DATA_BLOCK "DB2006_SA"
TITLE = DB2006_SA
{ S7_Optimized_Access := 'FALSE' }
AUTHOR : ABH
FAMILY : ZeusControl
VERSION : 1.0
//Bloique de datos Salida Analogica
   STRUCT
      SA { S7_SetPoint := 'False'} : Array[0.."N_MAX_DISP_SA"] of "UDT_ZC_DISP_SA";
      Mux { S7_SetPoint := 'False'} : Array[0.."N_MAX_MUX_DISP"] of "UDT_ZC_DISP_MUX_SA";
      Agrup : Array[0.."N_MAX_DISP_AGRUP"] of "UDT_ZC_DISP_AGRUP";
   END_STRUCT;


BEGIN
   SA[0].Hmi_Estado := 0;
   SA[0].Estado_ValorIngenieria := 0.0;
   SA[0].Estado_AutoMan := FALSE;
   SA[0].Estado_Enclavado := FALSE;
   SA[0].Alarmas_Min := FALSE;
   SA[0].Alarmas_Max := FALSE;
   SA[0].Alarmas_Escritura := FALSE;
   SA[0].Alarmas_Parametros := FALSE;
   SA[0].Alarmas_General := FALSE;
   SA[0].Config_Habilitar := FALSE;
   SA[0].Config_HabilitarAlarmaMin := FALSE;
   SA[0].Config_HabilitarAlarmaMax := FALSE;
   SA[0].Aux_oldAlarma := FALSE;
   SA[0].Aux_oldAutoMan := FALSE;
   SA[0].Estado_SeguridadOk := TRUE;
   SA[0].Config_GrupoAlarma := 0;
   SA[0].Aux_Estado := 0;
   SA[0].Estado_ValorTarjeta := 0;
   SA[0].Estado_Escritura := 16#0000;
   SA[0].Orden_ConsignaManual := 0.0;
   SA[0].Orden_ConsignaAuto := 0.0;
   SA[0].Orden_ConsignaEnclavado := 0.0;
   SA[0].Config_DireccionSalidaByte := 0;
   SA[0].Config_EscaladoMinTarjeta := 0;
   SA[0].Config_EscaladoMaxTarjeta := 27648;
   SA[0].Config_EscaladoMinIngenieria := 0.0;
   SA[0].Config_EscaladoMaxIngenieria := 0.0;
   SA[0].Config_EscaladoOffset := 0.0;
   SA[0].Config_ErrorMinIngenieria := 0.0;
   SA[0].Config_ErrorMaxIngenieria := 0.0;
   SA[1].Hmi_Estado := 1;
   SA[1].Estado_ValorIngenieria := 0.0;
   SA[1].Estado_AutoMan := FALSE;
   SA[1].Estado_Enclavado := FALSE;
   SA[1].Alarmas_Min := FALSE;
   SA[1].Alarmas_Max := FALSE;
   SA[1].Alarmas_Escritura := FALSE;
   SA[1].Alarmas_Parametros := FALSE;
   SA[1].Alarmas_General := FALSE;
   SA[1].Config_Habilitar := TRUE;
   SA[1].Config_HabilitarAlarmaMin := FALSE;
   SA[1].Config_HabilitarAlarmaMax := FALSE;
   SA[1].Aux_oldAlarma := FALSE;
   SA[1].Aux_oldAutoMan := FALSE;
   SA[1].Estado_SeguridadOk := TRUE;
   SA[1].Config_GrupoAlarma := 1;
   SA[1].Aux_Estado := 1;
   SA[1].Estado_ValorTarjeta := 0;
   SA[1].Estado_Escritura := 16#0000;
   SA[1].Orden_ConsignaManual := 0.0;
   SA[1].Orden_ConsignaAuto := 0.0;
   SA[1].Orden_ConsignaEnclavado := 0.0;
   SA[1].Config_DireccionSalidaByte := 2204;
   SA[1].Config_EscaladoMinTarjeta := 0;
   SA[1].Config_EscaladoMaxTarjeta := 27648;
   SA[1].Config_EscaladoMinIngenieria := 0.0;
   SA[1].Config_EscaladoMaxIngenieria := 100.0;
   SA[1].Config_EscaladoOffset := 0.0;
   SA[1].Config_ErrorMinIngenieria := 0.0;
   SA[1].Config_ErrorMaxIngenieria := 0.0;
   Mux[0].Habilitar := TRUE;
   Mux[0].ExisteCambio := FALSE;
   Mux[0].MaxVisible := FALSE;
   Mux[0].Index := 3;
   Mux[0].oldIndex := 3;
   Mux[0].SA.Hmi_Estado := 1;
   Mux[0].SA.Estado_ValorIngenieria := 0.0;
   Mux[0].SA.Estado_AutoMan := FALSE;
   Mux[0].SA.Estado_Enclavado := FALSE;
   Mux[0].SA.Alarmas_Min := FALSE;
   Mux[0].SA.Alarmas_Max := FALSE;
   Mux[0].SA.Alarmas_Escritura := FALSE;
   Mux[0].SA.Alarmas_Parametros := FALSE;
   Mux[0].SA.Alarmas_General := FALSE;
   Mux[0].SA.Config_Habilitar := TRUE;
   Mux[0].SA.Config_HabilitarAlarmaMin := FALSE;
   Mux[0].SA.Config_HabilitarAlarmaMax := FALSE;
   Mux[0].SA.Aux_oldAlarma := FALSE;
   Mux[0].SA.Aux_oldAutoMan := FALSE;
   Mux[0].SA.Estado_SeguridadOk := TRUE;
   Mux[0].SA.Config_GrupoAlarma := 1;
   Mux[0].SA.Aux_Estado := 1;
   Mux[0].SA.Estado_ValorTarjeta := 0;
   Mux[0].SA.Estado_Escritura := 16#0000;
   Mux[0].SA.Orden_ConsignaManual := 0.0;
   Mux[0].SA.Orden_ConsignaAuto := 0.0;
   Mux[0].SA.Orden_ConsignaEnclavado := 0.0;
   Mux[0].SA.Config_DireccionSalidaByte := 2208;
   Mux[0].SA.Config_EscaladoMinTarjeta := 0;
   Mux[0].SA.Config_EscaladoMaxTarjeta := 27648;
   Mux[0].SA.Config_EscaladoMinIngenieria := 0.0;
   Mux[0].SA.Config_EscaladoMaxIngenieria := 100.0;
   Mux[0].SA.Config_EscaladoOffset := 0.0;
   Mux[0].SA.Config_ErrorMinIngenieria := 0.0;
   Mux[0].SA.Config_ErrorMaxIngenieria := 0.0;
   Mux[1].Habilitar := TRUE;
   Mux[1].ExisteCambio := FALSE;
   Mux[1].MaxVisible := FALSE;
   Mux[1].Index := 0;
   Mux[1].oldIndex := 0;
   Mux[1].SA.Hmi_Estado := 0;
   Mux[1].SA.Estado_ValorIngenieria := 0.0;
   Mux[1].SA.Estado_AutoMan := FALSE;
   Mux[1].SA.Estado_Enclavado := FALSE;
   Mux[1].SA.Alarmas_Min := FALSE;
   Mux[1].SA.Alarmas_Max := FALSE;
   Mux[1].SA.Alarmas_Escritura := FALSE;
   Mux[1].SA.Alarmas_Parametros := FALSE;
   Mux[1].SA.Alarmas_General := FALSE;
   Mux[1].SA.Config_Habilitar := FALSE;
   Mux[1].SA.Config_HabilitarAlarmaMin := FALSE;
   Mux[1].SA.Config_HabilitarAlarmaMax := FALSE;
   Mux[1].SA.Aux_oldAlarma := FALSE;
   Mux[1].SA.Aux_oldAutoMan := FALSE;
   Mux[1].SA.Estado_SeguridadOk := TRUE;
   Mux[1].SA.Config_GrupoAlarma := 0;
   Mux[1].SA.Aux_Estado := 0;
   Mux[1].SA.Estado_ValorTarjeta := 0;
   Mux[1].SA.Estado_Escritura := 16#0000;
   Mux[1].SA.Orden_ConsignaManual := 0.0;
   Mux[1].SA.Orden_ConsignaAuto := 0.0;
   Mux[1].SA.Orden_ConsignaEnclavado := 0.0;
   Mux[1].SA.Config_DireccionSalidaByte := 0;
   Mux[1].SA.Config_EscaladoMinTarjeta := 0;
   Mux[1].SA.Config_EscaladoMaxTarjeta := 27648;
   Mux[1].SA.Config_EscaladoMinIngenieria := 0.0;
   Mux[1].SA.Config_EscaladoMaxIngenieria := 0.0;
   Mux[1].SA.Config_EscaladoOffset := 0.0;
   Mux[1].SA.Config_ErrorMinIngenieria := 0.0;
   Mux[1].SA.Config_ErrorMaxIngenieria := 0.0;
   Agrup[0].AlgunaEnManual := FALSE;
   Agrup[0].AlgunaAlarma := FALSE;
   Agrup[0].NuevaAlarma := FALSE;
   Agrup[1].AlgunaEnManual := FALSE;
   Agrup[1].AlgunaAlarma := FALSE;
   Agrup[1].NuevaAlarma := FALSE;

END_DATA_BLOCK

